{attribute 'qualified_only'}
VAR_GLOBAL
	stToHMI : ST_ToHMI;
	stFromHMI : ST_FromHMI; 
	iMenu : USINT;
	iPopupMenu : USINT;
END_VAR

(* stored: Version 1.1.0.1
   GVL HMI: Id {b4524cf6-01bd-4417-9a57-24146ccc07e2} *)
